Fanuc KAREL source: kt00146.KL

-- PROVISIONAL review KL for V940-1; original PC SHA256 302f9985f9e957065a97290694144fdee7d88f488f19c51a445d9eabdb047363
-- Incomplete behavior may be omitted. Consult companion uncertainty JSON. Do not deploy.
PROGRAM KT00146
%NOLOCKGROUP
VAR
  I2 : INTEGER
  OUT : REAL
-- UNRESOLVED_DECL Y1 type=002018
BEGIN
  -- V9_ZERO_TABLE_METADATA_HINT layout=0001; no indexed target words; source/name/runtime held
  -- UNRESOLVED_PC offsets 5-19; opcodes 2E,22,9D,33,B2
  -- UNRESOLVED_PC offsets 24-35; opcodes 2E,23
  -- UNRESOLVED_PC offsets 40-63; opcodes 22,9D,33,B1,21,55,64,23
  -- UNRESOLVED_PC offsets 68-72; opcodes 7F
END KT00146
